{attribute 'linkalways'} 
{attribute 'no_explicit_call' := 'This FB is a CLASS and must be accessed using methods or properties'}
{attribute 'enable_dynamic_creation'}
FUNCTION_BLOCK Node_RGBA_BLUE EXTENDS VisionNode
VAR
    out : _TcVnVector4_LREAL;
END_VAR

METHOD PUBLIC  Clone : I_Node
VAR
	pNode : POINTER TO Node_RGBA_BLUE;
END_VAR
pNode := __NEW(Node_RGBA_BLUE);
Clone := pNode^;
END_METHOD

METHOD FB_init : BOOL
VAR_INPUT
	bInitRetains : BOOL; // if TRUE, the retain variables are initialized (warm start / cold start)
	bInCopyCode : BOOL;  // if TRUE, the instance afterwards gets moved into the copy code (online change)
END_VAR
AddOutput('out', out);
END_METHOD

METHOD PROTECTED OnExecute : HRESULT
out.Value := GVL_COLOURS.RGBA_BLUE;
END_METHOD

METHOD PUBLIC PreExecutionCheck
VAR_INPUT
	Check : I_PreExecutionChecks;
END_VAR
END_METHOD

END_FUNCTION_BLOCK

(* stored: Version 1.1.0.1, ProductVersion 3.1.4024.13
   POU Node_RGBA_BLUE: Id {a6ad886e-06e3-0e36-2a02-a6ea273c1cfe}, SpecialFunc None
   Folder Constructor: Id {a3b9b697-4a9b-01a9-2fae-5034e9fe8ff7}
   Method Clone: Id {dd19f49f-08d3-06bb-2407-abdec321390b}
   Method FB_init: Id {c63eee60-7e18-01df-2f62-c4aa25778753}
   Method OnExecute: Id {8484f36f-a2e7-0d74-12af-1fd0257efb43}
   Method PreExecutionCheck: Id {ba813884-5fcd-0d41-355c-972d45ad8ebe} *)
